FUNCTION_BLOCK FB_AnalogInput
VAR_INPUT
	nRaw	:	INT;
	fEngMin :	REAL;
	fEngMax :	REAL;
END_VAR

VAR_OUTPUT
	fValue  :	REAL;
	bValid  :	BOOL;
END_VAR

VAR
	fRaw	:	REAL;
END_VAR

fRaw:= INT_TO_REAL(nRaw);

bValid := (nRaw >= 0);

IF bValid THEN
	fValue := fEngMin+(fRaw/32768.0)*(fEngMax -fEngMin);
ELSE
	fValue := fEngMin;
END_IF

END_FUNCTION_BLOCK

(* stored: Version 1.1.0.1, ProductVersion 3.1.4024.16
   POU FB_AnalogInput: Id {aecc98bf-0679-41be-99a7-fa4320218112}, SpecialFunc None *)
